FUNCTION_BLOCK FB_CarrierStop
VAR_INPUT
	Execute : BOOL;
END_VAR
VAR_OUTPUT
	Busy	: BOOL;
	Done	: BOOL;
	Error	: BOOL;
END_VAR
VAR
	_Decel : LREAL := 100000.0;

	X_AxisHalt	: MC_Halt;
	Z_AxisHalt	: MC_Halt;

	{attribute 'hide'}
	_X_Axis : POINTER TO AXIS_REF;
	{attribute 'hide'}
	_Z_Axis : POINTER TO AXIS_REF;

END_VAR

IF _X_Axis = 0 OR _Z_Axis = 0 THEN
	RETURN;
END_IF

X_AxisHalt(Axis			:= _X_Axis^,
			Deceleration := _Decel,
			Execute		:= Execute);

Z_AxisHalt(Axis			:= _Z_Axis^,
			Deceleration := _Decel,
			Execute		:= Execute);

Busy := X_AxisHalt.Busy OR Z_AxisHalt.Busy;

Done := X_AxisHalt.Done AND Z_AxisHalt.Done;

Error := X_AxisHalt.Error OR Z_AxisHalt.Error;

PROPERTY Decel : LREAL
GET
Decel := _Decel;
END_GET
SET
_Decel := Decel;
END_SET
END_PROPERTY

PROPERTY X_AxisRef : POINTER TO AXIS_REF
GET
X_AxisRef := _X_Axis;
END_GET
SET
_X_Axis := X_AxisRef;
END_SET
END_PROPERTY

PROPERTY Z_AxisRef : POINTER TO AXIS_REF
GET
Z_AxisRef := _Z_Axis;
END_GET
SET
_Z_Axis := Z_AxisRef;
END_SET
END_PROPERTY

END_FUNCTION_BLOCK

(* stored: Version 1.1.0.1, ProductVersion 3.1.4024.13
   POU FB_CarrierStop: Id {a062c842-c83b-4547-ab8a-140807b3c80c}, SpecialFunc None
   Property Decel: Id {080b320a-4ba7-4644-9ead-5e310b431ad5}
   Get Get: Id {12a8b3e8-589d-4813-bb88-6c0e410fd5ed}
   Set Set: Id {66c29c50-7ad3-4da2-ba25-d350335babfe}
   Property X_AxisRef: Id {c7b24212-2b13-4cd0-9843-8e793b748229}
   Get Get: Id {6401a6d1-7498-43f7-a188-0ea04789146e}
   Set Set: Id {808d9c69-d330-40e3-9002-cbaf2b20db18}
   Property Z_AxisRef: Id {a1ee128e-c87d-4a21-bd67-97a118d85bed}
   Get Get: Id {0198970b-9682-4c06-8cae-1dc08f3e872f}
   Set Set: Id {11f6ad41-b755-42c9-afb9-de9a0ec70674} *)
